# B&R Automation Studio project IecStringPrj (part 2)

#### test_float.c - Test IecStringFloat
```c
#include <UnitTest.h>
#include <IecString.h>
#include <string.h>
#include <stdint.h>
#include <float.h>

#define SAMPLE_SIZE 81
#define FULL_PRECISION 6
#define DEFAULT_WIDTH 0

_TEST test_float_variable(void) {
    char a[SAMPLE_SIZE];
    float value;
    int32_t status;

    value = 12e34f;

    status = IecStringFloat(a, sizeof(a), value,
                            DEFAULT_WIDTH, FULL_PRECISION, IECSTRING_FLAG_NONE);

    TEST_ASSERT_EQUAL_STRING("1.200000e+35", a);
    TEST_ASSERT_EQUAL_INT(IECSTRING_ERROR_NONE, status);

    TEST_DONE;
}

_TEST test_float_literal(void) {
    char a[SAMPLE_SIZE];
    int32_t status;

    status = IecStringFloat(a, sizeof(a), 12e34f,
                            DEFAULT_WIDTH, FULL_PRECISION, IECSTRING_FLAG_NONE);

    TEST_ASSERT_EQUAL_STRING("1.200000e+35", a);
    TEST_ASSERT_EQUAL_INT(IECSTRING_ERROR_NONE, status);

    TEST_DONE;
}

_TEST test_float_exponent_p5(void) {
    char a[SAMPLE_SIZE];
    int32_t status;

    status = IecStringFloat(a, sizeof(a), 123456.7f,
                            DEFAULT_WIDTH, FULL_PRECISION, IECSTRING_FLAG_NONE);

    TEST_ASSERT_EQUAL_STRING("123456.700000", a);
    TEST_ASSERT_EQUAL_INT(IECSTRING_ERROR_NONE, status);

    TEST_DONE;
}

_TEST test_float_exponent_p4(void) {
    char a[SAMPLE_SIZE];
    int32_t status;

    status = IecStringFloat(a, sizeof(a), 12345.67f,
                            DEFAULT_WIDTH, FULL_PRECISION, IECSTRING_FLAG_NONE);

    TEST_ASSERT_EQUAL_STRING("12345.670000", a);
    TEST_ASSERT_EQUAL_INT(IECSTRING_ERROR_NONE, status);

    TEST_DONE;
}

_TEST test_float_exponent_p3(void) {
    char a[SAMPLE_SIZE];
    int32_t status;

    status = IecStringFloat(a, sizeof(a), 1234.567f,
                            DEFAULT_WIDTH, FULL_PRECISION, IECSTRING_FLAG_NONE);

    TEST_ASSERT_EQUAL_STRING("1234.567000", a);
    TEST_ASSERT_EQUAL_INT(IECSTRING_ERROR_NONE, status);

    TEST_DONE;
}

_TEST test_float_exponent_p2(void) {
    char a[SAMPLE_SIZE];
    int32_t status;

    status = IecStringFloat(a, sizeof(a), 123.4567f,
                            DEFAULT_WIDTH, FULL_PRECISION, IECSTRING_FLAG_NONE);

    TEST_ASSERT_EQUAL_STRING("123.456700", a);
    TEST_ASSERT_EQUAL_INT(IECSTRING_ERROR_NONE, status);

    TEST_DONE;
}

_TEST test_float_exponent_p1(void) {
    char a[SAMPLE_SIZE];
    int32_t status;

    status = IecStringFloat(a, sizeof(a), 12.34567f,
                            DEFAULT_WIDTH, FULL_PRECISION, IECSTRING_FLAG_NONE);

    TEST_ASSERT_EQUAL_STRING("12.345670", a);
    TEST_ASSERT_EQUAL_INT(IECSTRING_ERROR_NONE, status);

    TEST_DONE;
}

_TEST test_float_exponent_0(void) {
    char a[SAMPLE_SIZE];
    int32_t status;

    status = IecStringFloat(a, sizeof(a), 1.234567f,
                            DEFAULT_WIDTH, FULL_PRECISION, IECSTRING_FLAG_NONE);

    TEST_ASSERT_EQUAL_STRING("1.234567", a);
    TEST_ASSERT_EQUAL_INT(IECSTRING_ERROR_NONE, status);

    TEST_DONE;
}

_TEST test_float_exponent_n1(void) {
    char a[SAMPLE_SIZE];
    int32_t status;

    status = IecStringFloat(a, sizeof(a), 0.1234567f,
                            DEFAULT_WIDTH, FULL_PRECISION, IECSTRING_FLAG_NONE);

    /* Rounding */
    TEST_ASSERT_EQUAL_STRING("0.123457", a);
    TEST_ASSERT_EQUAL_INT(IECSTRING_ERROR_NONE, status);

    TEST_DONE;
}

_TEST test_float_exponent_n2(void) {
    char a[SAMPLE_SIZE];
    int32_t status;

    status = IecStringFloat(a, sizeof(a), 0.01234567f,
                            DEFAULT_WIDTH, FULL_PRECISION, IECSTRING_FLAG_NONE);

    /* Rounding */
    TEST_ASSERT_EQUAL_STRING("0.012346", a);
    TEST_ASSERT_EQUAL_INT(IECSTRING_ERROR_NONE, status);

    TEST_DONE;
}

_TEST test_float_exponent_n3(void) {
    char a[SAMPLE_SIZE];
    int32_t status;

    status = IecStringFloat(a, sizeof(a), 0.001234567f,
                            DEFAULT_WIDTH, FULL_PRECISION, IECSTRING_FLAG_NONE);

    /* Rounding */
    TEST_ASSERT_EQUAL_STRING("0.001235", a);
    TEST_ASSERT_EQUAL_INT(IECSTRING_ERROR_NONE, status);

    TEST_DONE;
}

_TEST test_float_exponent_n4(void) {
    char a[SAMPLE_SIZE];
    int32_t status;

    status = IecStringFloat(a, sizeof(a), 0.0001234567f,
                            DEFAULT_WIDTH, FULL_PRECISION, IECSTRING_FLAG_NONE);

    TEST_ASSERT_EQUAL_STRING("0.000123", a);
    TEST_ASSERT_EQUAL_INT(IECSTRING_ERROR_NONE, status);

    TEST_DONE;
}

_TEST test_float_exponent_n5(void) {
    char a[SAMPLE_SIZE];
    int32_t status;

    status = IecStringFloat(a, sizeof(a), 0.00001234567f,
                            DEFAULT_WIDTH, FULL_PRECISION, IECSTRING_FLAG_NONE);

    TEST_ASSERT_EQUAL_STRING("0.000012", a);
    TEST_ASSERT_EQUAL_INT(IECSTRING_ERROR_NONE, status);

    TEST_DONE;
}

_TEST test_float_exponent_n6(void) {
    char a[SAMPLE_SIZE];
    int32_t status;

    status = IecStringFloat(a, sizeof(a), 0.000001234567f,
                            DEFAULT_WIDTH, FULL_PRECISION, IECSTRING_FLAG_NONE);

    TEST_ASSERT_EQUAL_STRING("0.000001", a);
    TEST_ASSERT_EQUAL_INT(IECSTRING_ERROR_NONE, status);

    TEST_DONE;
}

_TEST test_float_rollover_p5(void) {
    char a[SAMPLE_SIZE];
    int32_t status;

    /* Float stored as 999999.9375 or 1000000.0 */
    status = IecStringFloat(a, sizeof(a), 999999.97f,
                            DEFAULT_WIDTH, FULL_PRECISION, IECSTRING_FLAG_NONE);

    TEST_ASSERT_EQUAL_STRING("1.000000e+06", a);
    TEST_ASSERT_EQUAL_INT(IECSTRING_ERROR_NONE, status);

    TEST_DONE;
}

_TEST test_float_rollover_p2(void) {
    char a[SAMPLE_SIZE];
    int32_t status;

    /* Float stored as 999.99993896484375 or 1000.0 */
    status = IecStringFloat(a, sizeof(a), 999.99997f,
                            DEFAULT_WIDTH, FULL_PRECISION, IECSTRING_FLAG_NONE);

    TEST_ASSERT_EQUAL_STRING("1000.000000", a);
    TEST_ASSERT_EQUAL_INT(IECSTRING_ERROR_NONE, status);

    TEST_DONE;
}

_TEST test_float_rollover_0(void) {
    char a[SAMPLE_SIZE];
    int32_t status;

    status = IecStringFloat(a, sizeof(a), 0.9999995f,
                            DEFAULT_WIDTH, FULL_PRECISION, IECSTRING_FLAG_NONE);

    TEST_ASSERT_EQUAL_STRING("1.000000", a);
    TEST_ASSERT_EQUAL_INT(IECSTRING_ERROR_NONE, status);

    TEST_DONE;
}

_TEST test_float_rollover_n3(void) {
    char a[SAMPLE_SIZE];
    int32_t status;

    status = IecStringFloat(a, sizeof(a), 0.0009995f,
                            DEFAULT_WIDTH, FULL_PRECISION, IECSTRING_FLAG_NONE);

    TEST_ASSERT_EQUAL_STRING("0.001000", a);
    TEST_ASSERT_EQUAL_INT(IECSTRING_ERROR_NONE, status);

    TEST_DONE;
}

_TEST test_float_rollover_n6(void) {
    char a[SAMPLE_SIZE];
    int32_t status;

    /* Float stored as 9.99999883788e-07 or 9.99999997475e-07 */
    status = IecStringFloat(a, sizeof(a), 9.9999995e-7f,
                            DEFAULT_WIDTH, FULL_PRECISION, IECSTRING_FLAG_NONE);

    TEST_ASSERT_EQUAL_STRING("1.000000e-06", a);
    TEST_ASSERT_EQUAL_INT(IECSTRING_ERROR_NONE, status);

    TEST_DONE;
}

_TEST test_float_p37_A(void) {
    char a[SAMPLE_SIZE];
    int32_t status;

    /* Float representation is 9.99999460968e+37 */
    status = IecStringFloat(a, sizeof(a), 9.999995e37f,
                            DEFAULT_WIDTH, FULL_PRECISION, IECSTRING_FLAG_NONE);

    TEST_ASSERT_EQUAL_STRING("9.999995e+37", a);
    TEST_ASSERT_EQUAL_INT(IECSTRING_ERROR_NONE, status);

    TEST_DONE;
}

_TEST test_float_p37_B(void) {
    char a[SAMPLE_SIZE];
    int32_t status;

    /* Float representation is 9.99999866617e+37 or 9.99999968029e+37 */
    status = IecStringFloat(a, sizeof(a), 9.999999e37f,
                            DEFAULT_WIDTH, FULL_PRECISION, IECSTRING_FLAG_NONE);

    TEST_ASSERT_EQUAL_STRING("9.999999e+37", a);
    TEST_ASSERT_EQUAL_INT(IECSTRING_ERROR_NONE, status);

    TEST_DONE;
}

_TEST test_float_precision_3(void) {
    char a[SAMPLE_SIZE];
    int32_t status;

    status = IecStringFloat(a, sizeof(a), 0.123456f,
                            DEFAULT_WIDTH, 3, IECSTRING_FLAG_NONE);

    TEST_ASSERT_EQUAL_STRING("0.123", a);
    TEST_ASSERT_EQUAL_INT(IECSTRING_ERROR_NONE, status);

    TEST_DONE;
}

_TEST test_float_precision_3_round(void) {
    char a[SAMPLE_SIZE];
    int32_t status;

    status = IecStringFloat(a, sizeof(a), 0.99951f,
                            DEFAULT_WIDTH, 3, IECSTRING_FLAG_NONE);

    TEST_ASSERT_EQUAL_STRING("1.000", a);
    TEST_ASSERT_EQUAL_INT(IECSTRING_ERROR_NONE, status);

    TEST_DONE;
}

_TEST test_float_precision_0(void) {
    char a[SAMPLE_SIZE];
    int32_t status;

    status = IecStringFloat(a, sizeof(a), 123.456f,
                            DEFAULT_WIDTH, 0, IECSTRING_FLAG_NONE);

    TEST_ASSERT_EQUAL_STRING("123", a);
    TEST_ASSERT_EQUAL_INT(IECSTRING_ERROR_NONE, status);

    TEST_DONE;
}

_TEST test_float_precision_0_round(void) {
    char a[SAMPLE_SIZE];
    int32_t status;

    status = IecStringFloat(a, sizeof(a), 1.5f,
                            DEFAULT_WIDTH, 0, IECSTRING_FLAG_NONE);

    TEST_ASSERT_EQUAL_STRING("2", a);
    TEST_ASSERT_EQUAL_INT(IECSTRING_ERROR_NONE, status);

    TEST_DONE;
}

_TEST test_float_precision_0_notation(void) {
    char a[SAMPLE_SIZE];
    int32_t status;

    status = IecStringFloat(a, sizeof(a), 1.5e20f,
                            DEFAULT_WIDTH, 0, IECSTRING_FLAG_NONE);

    TEST_ASSERT_EQUAL_STRING("2e+20", a);
    TEST_ASSERT_EQUAL_INT(IECSTRING_ERROR_NONE, status);

    TEST_DONE;
}

_TEST test_float_max(void) {
    char a[SAMPLE_SIZE];
    int32_t status;

    status = IecStringFloat(a, sizeof(a), FLT_MAX,
                            DEFAULT_WIDTH, FULL_PRECISION, IECSTRING_FLAG_NONE);

    TEST_ASSERT_EQUAL_STRING("3.402823e+38", a);
    TEST_ASSERT_EQUAL_INT(IECSTRING_ERROR_NONE, status);

    TEST_DONE;
}

_TEST test_float_min(void) {
    char a[SAMPLE_SIZE];
    int32_t status;

    status = IecStringFloat(a, sizeof(a), FLT_MIN,
                            DEFAULT_WIDTH, FULL_PRECISION, IECSTRING_FLAG_NONE);

    TEST_ASSERT_EQUAL_STRING("1.175494e-38", a);
    TEST_ASSERT_EQUAL_INT(IECSTRING_ERROR_NONE, status);

    TEST_DONE;
}

_TEST test_float_zero(void) {
    char a[SAMPLE_SIZE];
    int32_t status, raw_value = 0;
    float value;

    memcpy(&value, &raw_value, 4);

    status = IecStringFloat(a, sizeof(a), value,
                            DEFAULT_WIDTH, FULL_PRECISION, IECSTRING_FLAG_NONE);

    TEST_ASSERT_EQUAL_STRING("0", a);
    TEST_ASSERT_EQUAL_INT(IECSTRING_ERROR_NONE, status);

    TEST_DONE;
}

_TEST test_float_negative_zero(void) {
    char a[SAMPLE_SIZE];
    int32_t status, raw_value = 0;
    float value;

    raw_value |= 1 << 31;
    memcpy(&value, &raw_value, 4);

    status = IecStringFloat(a, sizeof(a), value,
                            DEFAULT_WIDTH, FULL_PRECISION, IECSTRING_FLAG_NONE);

    TEST_ASSERT_EQUAL_STRING("-0", a);
    TEST_ASSERT_EQUAL_INT(IECSTRING_ERROR_NONE, status);

    TEST_DONE;
}

_TEST test_float_infinity(void) {
    char a[SAMPLE_SIZE];
    int32_t status, raw_value = 0;
    float value;

    raw_value |= 0xff << 23;
    memcpy(&value, &raw_value, 4);

    status = IecStringFloat(a, sizeof(a), value,
                            DEFAULT_WIDTH, FULL_PRECISION, IECSTRING_FLAG_NONE);

    TEST_ASSERT_EQUAL_STRING("inf", a);
    TEST_ASSERT_EQUAL_INT(IECSTRING_ERROR_NONE, status);

    TEST_DONE;
}

_TEST test_float_negative_infinity(void) {
    char a[SAMPLE_SIZE];
    int32_t status, raw_value = 0;
    float value;

    raw_value |= (1 << 31) + (0xff << 23);
    memcpy(&value, &raw_value, 4);

    status = IecStringFloat(a, sizeof(a), value,
                            DEFAULT_WIDTH, FULL_PRECISION, IECSTRING_FLAG_NONE);

    TEST_ASSERT_EQUAL_STRING("-inf", a);
    TEST_ASSERT_EQUAL_INT(IECSTRING_ERROR_NONE, status);

    TEST_DONE;
}

_TEST test_float_not_a_number(void) {
    char a[SAMPLE_SIZE];
    int32_t status, raw_value = 0;
    float value;

    raw_value |= (0xff << 23) + 1;
    memcpy(&value, &raw_value, 4);

    status = IecStringFloat(a, sizeof(a), value,
                            DEFAULT_WIDTH, FULL_PRECISION, IECSTRING_FLAG_NONE);

    TEST_ASSERT_EQUAL_STRING("NaN", a);
    TEST_ASSERT_EQUAL_INT(IECSTRING_ERROR_NONE, status);

    TEST_DONE;
}

_TEST test_float_size_zero(void) {
    char a[SAMPLE_SIZE];
    int32_t status;

    strcpy(a, "abc");
    status = IecStringFloat(a, 0, 123.0f,
                            DEFAULT_WIDTH, FULL_PRECISION, IECSTRING_FLAG_NONE);

    TEST_ASSERT_EQUAL_STRING("abc", a);
    TEST_ASSERT_EQUAL_INT(IECSTRING_ERROR_SIZE_ZERO, status);

    TEST_DONE;
}

_TEST test_float_size_one(void) {
    char a[SAMPLE_SIZE];
    int32_t status;

    strcpy(a, "abc");
    status = IecStringFloat(a, 1, 123.0f,
                            DEFAULT_WIDTH, FULL_PRECISION, IECSTRING_FLAG_NONE);

    TEST_ASSERT_EQUAL_STRING("", a);
    TEST_ASSERT_EQUAL_INT(IECSTRING_ERROR_SIZE_INVALID, status);

    TEST_DONE;
}

_TEST test_float_size_invalid(void) {
    char a[SAMPLE_SIZE];
    int32_t status;

    strcpy(a, "abc");
    /* Requires size of 11 for full precision 123.000000 */
    status = IecStringFloat(a, 6, 123.0f,
                            DEFAULT_WIDTH, FULL_PRECISION, IECSTRING_FLAG_NONE);

    TEST_ASSERT_EQUAL_STRING("", a);
    TEST_ASSERT_EQUAL_INT(IECSTRING_ERROR_SIZE_INVALID, status);

    TEST_DONE;
}

_TEST test_float_null(void) {
    int32_t status;

    status = IecStringFloat(NULL, SAMPLE_SIZE, 123.0f,
                            DEFAULT_WIDTH, FULL_PRECISION, IECSTRING_FLAG_NONE);

    TEST_ASSERT_EQUAL_INT(IECSTRING_ERROR_NULL, status);

    TEST_DONE;
}

UNITTEST_FIXTURES(fixtures) {
    new_TestFixture("IecStringFloat from variable", test_float_variable),
    new_TestFixture("IecStringFloat from literal", test_float_literal),
    new_TestFixture("IecStringFloat exponent +5", test_float_exponent_p5),
    new_TestFixture("IecStringFloat exponent +4", test_float_exponent_p4),
    new_TestFixture("IecStringFloat exponent +3", test_float_exponent_p3),
    new_TestFixture("IecStringFloat exponent +2", test_float_exponent_p2),
    new_TestFixture("IecStringFloat exponent +1", test_float_exponent_p1),
    new_TestFixture("IecStringFloat exponent  0", test_float_exponent_0),
    new_TestFixture("IecStringFloat exponent -1", test_float_exponent_n1),
    new_TestFixture("IecStringFloat exponent -2", test_float_exponent_n2),
    new_TestFixture("IecStringFloat exponent -3", test_float_exponent_n3),
    new_TestFixture("IecStringFloat exponent -4", test_float_exponent_n4),
    new_TestFixture("IecStringFloat exponent -5", test_float_exponent_n5),
    new_TestFixture("IecStringFloat exponent -6", test_float_exponent_n6),
    new_TestFixture("IecStringFloat rollover +5", test_float_rollover_p5),
    new_TestFixture("IecStringFloat rollover +2", test_float_rollover_p2),
    new_TestFixture("IecStringFloat rollover  0", test_float_rollover_0),
    new_TestFixture("IecStringFloat rollover -3", test_float_rollover_n3),
    new_TestFixture("IecStringFloat rollover -6", test_float_rollover_n6),
    new_TestFixture("IecStringFloat precision 3", test_float_precision_3),
    new_TestFixture("IecStringFloat precision 3 round",
                    test_float_precision_3_round),
    new_TestFixture("IecStringFloat exponent +37 test A", test_float_p37_A),
    new_TestFixture("IecStringFloat exponent +37 test B", test_float_p37_B),
    new_TestFixture("IecStringFloat precision 0", test_float_precision_0),
    new_TestFixture("IecStringFloat precision 0 round",
                    test_float_precision_0_round),
    new_TestFixture("IecStringFloat precision 0 scientific notation",
                    test_float_precision_0_notation),
    new_TestFixture("IecStringFloat max", test_float_max),
    new_TestFixture("IecStringFloat min", test_float_min),
    new_TestFixture("IecStringFloat zero", test_float_zero),
    new_TestFixture("IecStringFloat negative zero", test_float_negative_zero),
    new_TestFixture("IecStringFloat infinity", test_float_infinity),
    new_TestFixture("IecStringFloat negative infinity",
                    test_float_negative_infinity),
    new_TestFixture("IecStringFloat not a number", test_float_not_a_number),
    new_TestFixture("IecStringFloat size zero", test_float_size_zero),
    new_TestFixture("IecStringFloat size one", test_float_size_one),
    new_TestFixture("IecStringFloat size invalid", test_float_size_invalid),
    new_TestFixture("IecStringFloat null", test_float_null)
};

UNITTEST_CALLER_TEST(float_set, "IecStringFloat test set", fixtures);
```

#### test_date_time.c - Test IecStringDateTime
```c
#include <UnitTest.h>
#include <IecString.h>
#include <astime.h>
#include <string.h>
#include <stdint.h>

#define SAMPLE_SIZE 81

DTStructure value = {
    .year = 2024,
    .month = 1,
    .day = 9,
    .wday = 2,
    .hour = 13,
    .minute = 4,
    .second = 9,
    .millisec = 55
};

_TEST test_date_time_default(void) {
    char a[SAMPLE_SIZE];
    int32_t status;

    status = IecStringDateTime(a, sizeof(a), &value, NULL);

    TEST_ASSERT_EQUAL_STRING("2024-01-09 13:04", a);
    TEST_ASSERT_EQUAL_INT(IECSTRING_ERROR_NONE, status);

    TEST_DONE;
}

_TEST test_date_time_formal_date(void) {
    char a[SAMPLE_SIZE];
    int32_t status;

    status = IecStringDateTime(a, sizeof(a), &value, "dddd, MMMM d, yyyy");

    TEST_ASSERT_EQUAL_STRING("Tuesday, January 9, 2024", a);
    TEST_ASSERT_EQUAL_INT(IECSTRING_ERROR_NONE, status);

    TEST_DONE;
}

UNITTEST_FIXTURES(fixtures) {
    new_TestFixture("IecStringDateTime default", test_date_time_default),
    new_TestFixture("IecStringDateTime formal date", test_date_time_formal_date)
};

UNITTEST_CALLER_TEST(date_time_set, "IecStringDateTime test set", fixtures);
```

#### test_integer.c - not listed in the package file held
```c
#include <UnitTest.h>
#include <IecString.h>
#include <string.h>
#include <stdint.h>

_TEST test_integer_zeros(void) {
    char a[81];
    int32_t number, status;

    number = 1234;

    status = IecStringInteger(a, sizeof(a), number, 6, '0');

    TEST_ASSERT_EQUAL_STRING("001234", a);
    TEST_ASSERT_EQUAL_INT(0, status);

    TEST_DONE;
}

_TEST test_integer_spaces(void) {
    char a[81];
    int32_t number, status;

    number = -5678;

    status = IecStringInteger(a, sizeof(a), number, 6, ' ');

    /* Width includes sign */
    TEST_ASSERT_EQUAL_STRING("- 5678", a);
    TEST_ASSERT_EQUAL_INT(0, status);

    /* Defaults to spaces */
    status = IecStringInteger(a, sizeof(a), number, 6, 0);

    TEST_ASSERT_EQUAL_STRING("- 5678", a);
    TEST_ASSERT_EQUAL_INT(0, status);

    TEST_DONE;
}

_TEST test_integer_tilde(void) {
    char a[81];
    int32_t number, status;

    number = 9012;

    status = IecStringInteger(a, sizeof(a), number, 6, '~');

    TEST_ASSERT_EQUAL_STRING("~~9012", a);
    TEST_ASSERT_EQUAL_INT(0, status);

    TEST_DONE;
}

_TEST test_integer_max(void) {
    char a[81];
    int32_t number, status;

    number = INT32_MAX;

    status = IecStringInteger(a, sizeof(a), number, 0, '0');

    TEST_ASSERT_EQUAL_STRING("2147483647", a);
    TEST_ASSERT_EQUAL_INT(0, status);

    TEST_DONE;
}

_TEST test_integer_min(void) {
    char a[81];
    int32_t number, status;

    number = INT32_MIN;

    status = IecStringInteger(a, sizeof(a), number, 0, '0');

    TEST_ASSERT_EQUAL_STRING("-2147483648", a);
    TEST_ASSERT_EQUAL_INT(0, status);

    TEST_DONE;
}

_TEST test_integer_size(void) {
    char a[6];
    int32_t number, status;

    strcpy(a, "abc");
    number = 123456;

    status = IecStringInteger(a, sizeof(a), number, 0, '0');

    TEST_ASSERT_EQUAL_STRING("abc", a);
    TEST_ASSERT_EQUAL_INT(IECSTRING_ERROR_SIZE, status);

    TEST_DONE;
}

_TEST test_integer_null(void) {
    int32_t number, status;

    number = 123456;

    status = IecStringInteger(NULL, 7, number, 0, '0');

    TEST_ASSERT_EQUAL_INT(IECSTRING_ERROR_NULL, status);

    TEST_DONE;
}

UNITTEST_FIXTURES(fixtures) {
    new_TestFixture("IecStringInteger zeros", test_integer_zeros),
    new_TestFixture("IecStringInteger spaces", test_integer_spaces),
    new_TestFixture("IecStringInteger tilde", test_integer_tilde),
    new_TestFixture("IecStringInteger max", test_integer_max),
    new_TestFixture("IecStringInteger min", test_integer_min),
    new_TestFixture("IecStringInteger size error", test_integer_size),
    new_TestFixture("IecStringInteger null error", test_integer_null)
};

UNITTEST_CALLER_TEST (padint_set, "IecStringInteger test set", fixtures);
```

### Program Logical/Source/UnitTest/TestFloat (ANSIC)

#### Variables.var
```iecst
VAR
	FloatValue : REAL;
	PromotionToDouble : LREAL;
	LibFloatText : STRING[80];
	BrsFloatText : STRING[80];
	FloatRaw : UDINT;
	TestInfinity : BOOL;
	TestNotANumber : BOOL;
	Log10Value : REAL;
	Precision : USINT;
END_VAR
```

#### Main.c
```c
#include <bur/plc.h>
#include <Variablesvar.h>
#include <IecString.h>
#include <AsBrStr.h>
#include <stdint.h>
#include <math.h>

void _CYCLIC ProgramCyclic(void) {
    IecStringFloat(LibFloatText, sizeof(LibFloatText), FloatValue);
    brsftoa(FloatValue, (uint32_t)BrsFloatText);
    PromotionToDouble = FloatValue;
    FloatRaw = *(uint32_t*)&FloatValue;

    if (TestInfinity) {
        TestInfinity = 0;
        FloatValue *= 1.0e38f;
    }

    if (TestNotANumber) {
        TestNotANumber = 0;
        FloatValue /= 0.0f;
    }

    Log10Value = log10f(FloatValue);
}
```

### Program Logical/Source/UnitTest/TestCopy (ANSIC)

#### Variables.var
```iecst
VAR
	String1 : STRING[80];
	String2 : STRING[80];
	MySize : UDINT := 6;
	MyStatus : DINT;
END_VAR
```

#### Main.c
```c
#include <bur/plc.h>
#include <Variablesvar.h>
#include <IecString.h>

void _CYCLIC ProgramCyclic(void) {
    MyStatus = IecStringCopy(String1, MySize, String2);
}
```

### Program Logical/Source/UnitTest/TestDT (IEC)

#### Variables.var
```iecst
VAR
	DateAndTimeData : DTStructure;
	String1 : STRING[80];
	String2 : STRING[80];
	GetDateAndTime : DTStructureGetTime;
END_VAR
```

#### Main.st
```iecst
PROGRAM _INIT
	GetDateAndTime(enable := TRUE, pDTStructure := ADR(DateAndTimeData));
END_PROGRAM

PROGRAM _CYCLIC
	IecStringDateTime(String1, SIZEOF(String1), DateAndTimeData, String2);
END_PROGRAM
```

### Program Logical/Source/Example/ExSplit (IEC)

#### Variables.var
```iecst
(*Command*)
VAR
	Run : BOOL;
END_VAR
(*Data*)
VAR
	Source : STRING[80];
	SourceReference : REFERENCE TO STRING[80];
	NextAddress : UDINT;
	Delimeters : STRING[80];
	Words : ARRAY[0..9] OF STRING[80];
	Index : USINT;
END_VAR
```

#### Main.st
```iecst
PROGRAM _INIT

	Source := 'The quick brown fox jumps over the lazy dog';
	Delimeters := ' ';

END_PROGRAM

PROGRAM _CYCLIC

	IF Run THEN
		Run := FALSE;

		brsmemset(ADR(Words), 0, SIZEOF(Words));
		Index := 0;

		SourceReference ACCESS ADR(Source);
		REPEAT
			IecStringSplit(Words[Index], SIZEOF(Words[Index]), SourceReference, Delimeters, NextAddress);
			SourceReference ACCESS NextAddress;
			Index := Index + 1;
		UNTIL
			Index >= SIZEOF(Words) / SIZEOF(Words[0]) OR NextAddress = 0
		END_REPEAT
		SourceReference ACCESS ADR(Source);
	END_IF

END_PROGRAM
```

### Program Logical/Source/Performance/ACopy1C (ANSIC) - Performance of strcpy

#### Main.c
```c
#include <bur/plc.h>
#include <string.h>

void _CYCLIC ProgramCyclic(void)
{
    char a[81];
    int i;
    for (i = 0; i < 100; i++)
        strcpy(a, "This is a test of string copy performance across multiple libraries.");
}
```

### Program Logical/Source/Performance/ACopy2Iec (IEC) - Performacce of IEC string assignment

#### Variables.var
```iecst
VAR
	i : INT;
	a : STRING[254];
	b : STRING[254] := '0123456789abcdefghij0123456789abcdefghij0123456789abcdefghij0123456789abcdefghij';
END_VAR
```

#### Main.st
```iecst
(* 100 calls to copy 80 characters *)
PROGRAM _CYCLIC
	FOR i := 0 TO 99 DO
		a := b;
	END_FOR
END_PROGRAM
```

### Program Logical/Source/Performance/ACopy3Brs (ANSIC) - Performance of brsstrcpy

#### Main.c
```c
#include <bur/plc.h>
#include <AsBrStr.h>

char a[255];
int i;

/* 100 calls to copy 80 characters */
void _CYCLIC ProgramCyclic(void)
{
    for (i = 0; i < 100; i++)
    {
        brsstrcpy((unsigned long)a,
                  (unsigned long)"0123456789abcdefghij0123456789abcdefghij"
                                 "0123456789abcdefghij0123456789abcdefghij");
    }
}
```

### Program Logical/Source/Performance/ACopy4Lib (ANSIC) - Performance of IecStringCopy

#### Main.c
```c
#include <bur/plc.h>
#include <IecString.h>

char a[255];
int i;

/* 100 calls to copy 80 characters */
void _CYCLIC ProgramCyclic(void)
{
    for (i = 0; i < 100; i++)
    {
        IecStringCopy(a, sizeof(a), "0123456789abcdefghij0123456789abcdefghij"
                                    "0123456789abcdefghij0123456789abcdefghij");
    }
}
```

### Program Logical/Source/Performance/BCat1C (ANSIC) - Performance of strcat

#### Main.c
```c
#include <bur/plc.h>
#include <string.h>

char a[255] = "Hello World! 1234567890.";
int i;

void _CYCLIC ProgramCyclic(void) {
    for (i = 0; i < 100; i++) {
        a[24] = '\0';
        strcat(a, " The quick brown fox jumps over the lazy dog.");
    }
}
```

### Program Logical/Source/Performance/BCat2Iec (IEC) - Performance of CONCAT

#### Variables.var
```iecst
VAR
	i : INT;
	a : STRING[255];
END_VAR
```

#### Main.st
```iecst
(* 100 calls to concatenate 80 characters to length of 80 *)
PROGRAM _CYCLIC
	FOR i := 0 TO 99 DO
		a := CONCAT('0123456789abcdefghij0123456789abcdefghij0123456789abcdefghij0123456789abcdefghij', '0123456789abcdefghij0123456789abcdefghij0123456789abcdefghij0123456789abcdefghij');
	END_FOR
END_PROGRAM
```

### Program Logical/Source/Performance/BCat3Brs (ANSIC) - Performance of brsstrcat

#### Main.c
```c
#include <bur/plc.h>
#include <AsBrStr.h>
#include <stdint.h>

char a[81] = "Hello World! 1234567890.";
int i;

void _CYCLIC ProgramCyclic(void) {
    for (i = 0; i < 100; i++) {
        a[24] = '\0';
        brsstrcat((uint32_t)a, (uint32_t)" The quick brown fox jumps over the lazy dog.");
    }
}
```

### Program Logical/Source/Performance/BCat4Lib (ANSIC) - Performance of IecStringConcat

#### Main.c
```c
#include <bur/plc.h>
#include <IecString.h>

char a[255] = "0123456789abcdefghij0123456789abcdefghij"
              "0123456789abcdefghij0123456789abcdefghij";
int i;

/* 100 calls to concatenate 80 characters to length of 80 */
void _CYCLIC ProgramCyclic(void)
{
    for (i = 0; i < 100; i++)
    {
        a[80] = '\0';
        IecStringConcat(a, sizeof(a),
                        "0123456789abcdefghij0123456789abcdefghij"
                        "0123456789abcdefghij0123456789abcdefghij");
    }
}
```

### Program Logical/Source/Performance/EDec2Iec (IEC) - Performance of DINT_TO_STRING

#### Variables.var
```iecst
VAR
	i : INT;
	number : DINT := -2001001001;
	a : STRING[20];
END_VAR
```

#### Main.st
```iecst
(* 100 calls to convert integer to string *)
PROGRAM _CYCLIC
	FOR i := 0 TO 99 DO
		a := DINT_TO_STRING(number);
	END_FOR
END_PROGRAM
```

### Program Logical/Source/Performance/EDec3Brs (ANSIC) - Performance of brsitoa

#### Main.c
```c
#include <bur/plc.h>
#include <AsBrStr.h>

char a[21];
int i;
const signed long number = -2001001001;

void _CYCLIC ProgramCyclic(void) {
    for (i = 0; i < 100; i++)
        brsitoa(number, (unsigned long)a);
}
```

### Program Logical/Source/Performance/EDec4Lib (ANSIC) - Performance of IecStringDecimal

#### Main.c
```c
#include <bur/plc.h>
#include <IecString.h>

char a[21];
int i;
const signed long number = -2001001001;

void _CYCLIC ProgramCyclic(void) {
    for (i = 0; i < 100; i++)
        IecStringDecimal(a, sizeof(a), number, 5, '0', 0);
}
```

### Program Logical/Source/Performance/FFp2Iec (IEC) - Performance of AsIecCon's REAL_TO_STRING

#### Main.st
```iecst
(* 100 calls to convert float to string *)
PROGRAM _CYCLIC
	FOR i := 0 TO 99 DO
		a := REAL_TO_STRING(123.456e-23);
	END_FOR
END_PROGRAM
```

### Program Logical/Source/Performance/FFp3Brs (ANSIC) - Performance of AsBrStr's brsftoa

#### Main.c
```c
#include <bur/plc.h>
#include <AsBrStr.h>

char a[81];
int i;

/* 100 calls to convert float to string */
void _CYCLIC ProgramCyclic(void)
{
    for (i = 0; i < 100; i++)
        brsftoa(123.456e-23f, (unsigned long)a);
}
```

### Program Logical/Source/Performance/FFp4Lib (ANSIC) - Performance of IecStringFloat

#### Main.c
```c
#include <bur/plc.h>
#include <IecString.h>

char a[81];
int i;

/* 100 calls to convert float to string */
void _CYCLIC ProgramCyclic(void)
{
    for (i = 0; i < 100; i++)
        IecStringFloat(a, sizeof(a), 123.456e-23f, 0, 6, IECSTRING_FLAG_NONE);
}
```

### Program Logical/Source/Performance/ACopy2Br

#### Main.c
```c
#include <bur/plc.h>
#include <stdint.h>
#include <AsBrStr.h>

void _CYCLIC ProgramCyclic(void)
{
    char a[81];
    int i;
    for (i = 0; i < 100; i++)
        brsstrcpy((uint32_t)a, (uint32_t)"This is a test of string copy performance across multiple libraries");
}
```

### Program Logical/Source/Performance/ACopy3IS (ANSIC)

#### Main.c - Init, cyclic, exit code
```c
#include <bur/plc.h>
#include <IecString.h>

void _CYCLIC ProgramCyclic(void)
{
    char a[81];
    int i;
    for (i = 0; i < 100; i++)
        IecStringCopy(a, sizeof(a), "This is a test of string copy performance");
}
```

### Program Logical/Source/Performance/BCat2Br

#### Main.c
```c
#include <bur/plc.h>
#include <AsBrStr.h>
#include <stdint.h>

void _CYCLIC ProgramCyclic(void)
{
    char a[81] = "Hello World! 1234567890.";
    int i;
    for (i = 0; i < 100; i++) {
        a[19] = '\0';
        brsstrcat((uint32_t)a, (uint32_t)" The quick brown fox jumps over the lazy dog.");
    }
}
```

### Program Logical/Source/Performance/BCat3IS

#### Main.c
```c
#include <bur/plc.h>
#include <IecString.h>

void _CYCLIC ProgramCyclic(void)
{
    char a[81] = "Hello World! 1234567890.";
    int i;
    for (i = 0; i < 100; i++) {
        a[19] = '\0';
        IecStringConcat(a, sizeof(a), " The quick brown fox jumps over the lazy dog.");
    }
}
```

### Program Logical/Source/Performance/CPUCopy

#### Main.c
```c
#include <bur/plc.h>
#include <bur/plctypes.h>
#include <IecString.h>
#include <AsBrStr.h>
#include <string.h>

_LOCAL UINT count _VAR_INIT(100);

void _CYCLIC ProgramCyclic(void)
{
    char a[81], b[81];
    DINT i;
    IecStringCopy(b, sizeof(b), "This is a test of string copy performance");

    /* Test strcpy */
    for (i = 0; i < count; i++)
        strcpy(a, b);

    /* Test brsstrcpy */
    for (i = 0; i < count; i++)
        brsstrcpy((UDINT)a, (UDINT)b);

    /* Test IecStringCopy */
    for (i = 0; i < count; i++)
        IecStringCopy(a, sizeof(a), b);
}
```

### Program Logical/Source/Performance/CPUDecimal

#### Main.c
```c
#include <bur/plc.h>
#include <bur/plctypes.h>
#include <IecString.h>
#include <AsBrStr.h>

_LOCAL UINT count _VAR_INIT(100);

void _CYCLIC ProgramCyclic(void)
{
    char a[21];
    DINT i, number = -2001001001;

    /* Test brsitoa */
    for (i = 0; i < count; i++)
        brsitoa(number, (UDINT)a);

    /* Test IecStringInteger */
    for (i = 0; i < count; i++)
        IecStringInteger(a, sizeof(a), number, 5, '0');
}
```

### Program Logical/Source/Performance/EDec2Br

#### Main.c
```c
#include <bur/plc.h>
#include <stdint.h>
#include <AsBrStr.h>

void _CYCLIC ProgramCyclic(void)
{
    char a[21];
    int32_t i, number = -2001001001;
    for (i = 0; i < 100; i++)
        brsitoa(number, (UDINT)a);
}
```

### Program Logical/Source/Performance/PerfBase

#### Main.c
```c
#include <bur/plc.h>

void _CYCLIC ProgramCyclic(void)
{
    char a[81], b[81];
    int i;
    for (i = 0; i < 100; i++)
        i;
}
```

### Program Logical/Source/Performance/PerfBrCopy

#### Main.c
```c
#include <bur/plc.h>
#include <bur/plctypes.h>
#include <AsBrStr.h>

void _CYCLIC ProgramCyclic(void)
{
    char a[81];
    int i;
    for (i = 0; i < 100; i++)
        brsstrcpy((UDINT)a, "This is a test of string copy performance");
}
```

### Program Logical/Source/Performance/PerfISDec

#### Main.c
```c
#include <bur/plc.h>
#include <stdint.h>
#include <IecString.h>

void _CYCLIC ProgramCyclic(void)
{
    char a[21];
    int32_t i, number = -2001001001;
    for (i = 0; i < 100; i++)
        IecStringInteger(a, sizeof(a), number, 5, '0');
}
```

### Program Logical/Source/Compare/CFloat (ANSIC) - Test floating point values

#### Main.c
```c
#include <bur/plc.h>
#include <stdint.h>
#include <string.h>

_LOCAL float number;
_LOCAL uint32_t data, sign, exponent, fraction;
_LOCAL int32_t int_cast;

void _CYCLIC ProgramCyclic(void)
{
    memcpy(&data, &number, sizeof(data));
    sign = (data >> 31) & 0x1;
    exponent = (data >> 23) & 0xFF;
    fraction = data & 0x7FFFFF;
    int_cast = (int)number;
}
```

### Program Logical/Source/Compare/Float (IEC)

#### Variables.var
```iecst
VAR
	FloatValue : REAL;
	DoublePromotionValue : LREAL;
	LibFloatText : STRING[80];
	BrsFloatText : STRING[80];
END_VAR
```

#### Main.st
```iecst
PROGRAM _CYCLIC
	DoublePromotionValue := FloatValue;
	IecStringFloat(LibFloatText, SIZEOF(LibFloatText), FloatValue);
	brsftoa(FloatValue, ADR(BrsFloatText));
END_PROGRAM
```

### Program Logical/Source/Compare/BrDecimal

#### Variables.var
```iecst
VAR
	Number : DINT;
	NumberText : STRING[14];
	NumberData : REFERENCE TO ARRAY[0..14] OF USINT;
END_VAR
```

#### Main.st
```iecst
PROGRAM _CYCLIC

	brsitoa(Number, ADR(NumberText));
	NumberData ACCESS ADR(NumberText);

END_PROGRAM
```

### Program Logical/Source/Compare/BrFloat

#### Variables.var
```iecst
VAR
	Number : REAL;
	NumberText : STRING[14];
	NumberData : REFERENCE TO ARRAY[0..14] OF USINT;
END_VAR
```

#### Main.st
```iecst
PROGRAM _CYCLIC

	brsftoa(Number, ADR(NumberText));
	NumberData ACCESS ADR(NumberText);

END_PROGRAM
```

### Program Logical/Source/Sample/IECST (IEC)

#### Variables.var
```iecst
(*IecStringCopy*)
VAR
	Source : STRING[10] := 'Program';
	Destination : STRING[5];
END_VAR
(*IecStringFormat*)
VAR
	FromattedString : STRING[80];
	FormatValues : IecStringFormatType;
END_VAR
(*IecStringInteger*)
VAR
	MyInteger : INT;
	PaddedInteger : STRING[80];
END_VAR
(*IecStringDateTime*)
VAR
	DateTimeString : STRING[80];
	FormatDateTime : STRING[80];
	DateTime : DTStructure;
	GetDateTime : DTStructureGetTime;
	CurrentDateTime : DTStructure;
END_VAR
(*Raw characters*)
VAR
	Raw1 : ARRAY[0..10] OF USINT;
	Raw2 : ARRAY[0..10] OF USINT;
	ReferenceString1 : REFERENCE TO STRING[10];
	ReferenceString2 : REFERENCE TO STRING[10];
END_VAR
```

#### Main.st
```iecst
PROGRAM _INIT

	FormatValues.b[0] := TRUE;
	FormatValues.f[0] := 12.34;
	FormatValues.i[0] := 33;
	FormatValues.s[0] := 'All Clear';

END_PROGRAM

PROGRAM _CYCLIC

	IecStringCopy(Destination,
		SIZEOF(Destination),
		Source);

	ReferenceString1 ACCESS ADR(Raw1);
	ReferenceString2 ACCESS ADR(Raw2);
	IecStringCopy(ReferenceString1, SIZEOF(ReferenceString1), ReferenceString2);

	IecStringFormat(FromattedString,
		SIZEOF(FromattedString),
		'Error: %b, Temp: %f C, Step: %i, Message: %s',
		FormatValues);

	IecStringInteger(PaddedInteger,
		SIZEOF(PaddedInteger),
		MyInteger,
		6,
		FALSE);

	GetDateTime(enable := TRUE, pDTStructure := ADR(CurrentDateTime));
	IecStringDateTime(DateTimeString, SIZEOF(DateTimeString), FormatDateTime, DateTime);

END_PROGRAM
```

### Program Logical/Source/Sample/Float (IEC)

#### Variables.var
```iecst
VAR
	String1 : STRING[80];
	Value : REAL;
	Width : USINT;
	Precision : USINT;
END_VAR
```

#### Main.st
```iecst
PROGRAM _CYCLIC

	IecStringFloat(String1, SIZEOF(String1), Value, Width, Precision, IECSTRING_FLAG_NONE);

END_PROGRAM
```

### Program Logical/Source/Sample/ExFloat

#### Variables.var
```iecst
VAR
	Float : REAL;
	FloatText : STRING[80];
END_VAR
```

#### Main.st
```iecst
PROGRAM _CYCLIC

	IecStringFloat(FloatText, SIZEOF(FloatText), Float);

END_PROGRAM
```

- IecStringText.csv (not shown)

- IecStringGenerate.py (not shown)

### Program Logical/CUsage

#### Variables.var
```iecst
VAR
	format : STRING[80];
	formatArgs : FormatStringArgumentsType;
	message : STRING[80];
	length : UDINT;
END_VAR
(*Pad whole number*)
VAR
	myNumber : DINT;
	number : STRING[20];
	digits : USINT;
	spaces : BOOL;
END_VAR
```

#### Main.c
```c
#include <bur/plctypes.h>

#ifdef _DEFAULT_INCLUDES
	#include <AsDefault.h>
#endif

#include <stdbool.h>
#include <string.h>

void _INIT ProgramInit(void)
{
	// Runtime values
	formatArgs.b[0] = false; // BOOL
	formatArgs.r[0] = 78.768; // LREAL
	formatArgs.i[0] = -2144327918; // DINT, e.g. Status ID
	strcpy(formatArgs.s[0], "INIT"); // STRING

	strcpy(format, "Status %b, Temp %r F, Code %i, State %s");

	myNumber = -1234;
	digits = 6;
	spaces = false;
}

void _CYCLIC ProgramCyclic(void)
{
	length = IecFormatString(message, sizeof(message), format, &formatArgs);

	IecPadNumber(myNumber, number, digits, spaces);
}

void _EXIT ProgramExit(void)
{

}
```

### Program Logical/IECST

#### Variables.var
```iecst
(*IecStringCopy*)
VAR
	Source : STRING[10] := 'Program';
	Destination : STRING[5];
END_VAR
(*IecStringFormat*)
VAR
	FromattedString : STRING[80];
	FormatValues : IecStringFormatType;
END_VAR
(*IecStringInteger*)
VAR
	MyInteger : INT;
	PaddedInteger : STRING[80];
END_VAR
(*IecStringDateTime*)
VAR
	DateTimeString : STRING[80];
	FormatDateTime : STRING[80];
END_VAR
```

#### Main.st
```iecst
PROGRAM _INIT

	FormatValues.b[0] := TRUE;
	FormatValues.f[0] := 12.34;
	FormatValues.i[0] := 33;
	FormatValues.s[0] := 'All Clear';

END_PROGRAM

PROGRAM _CYCLIC

	IecStringCopy(Destination,
		SIZEOF(Destination),
		Source);

	IecStringFormat(FromattedString,
		SIZEOF(FromattedString),
		'Error: %b, Temp: %f C, Step: %i, Message: %s',
		FormatValues);

	IecStringInteger(PaddedInteger,
		SIZEOF(PaddedInteger),
		MyInteger,
		6,
		FALSE);

	GetDateTime(enable := TRUE, pDTStructure := ADR(CurrentDateTime));
	IecStringDateTime(DateTimeString, SIZEOF(DateTimeString), FormatDateTime, DateTime);

END_PROGRAM
```

### Program Logical/Program

#### Variables.var
```iecst
VAR
	AllocationReturnStatus : UDINT;
	CyclicReturnStatus : UDINT;
	FreeReturnStatus : UDINT;
END_VAR
VAR CONSTANT
	STR_LEN_ALARM_MSG : USINT := 125;
END_VAR
VAR
	sConstructMessage : STRING[STR_LEN_ALARM_MSG];
	sFormattedMessage : STRING[STR_LEN_ALARM_MSG];
	MessageArguments : FormatStringArgumentsType;
	CmdLog : BOOL;
	EventID : DINT;
	ErrorCode : UINT;
END_VAR
```

#### Main.st
```iecst
(*******************************************************************************
 * Copyright: B&R Industrial Automation
 * Author:    Tyler Matijevich
 * Created:   September 27, 2020/11:19
********************************************************************************
 * Description: Example program for formatting string in IEC code and logging
 user entries in the logger
********************************************************************************)

PROGRAM _INIT

	// Allocates the FIFO buffer for the logger
	AllocationReturnStatus := BRSE_ARL_Alloc(ID := 1, Name := 'AppLog', LogbookSize := 10000, MessageSize := STR_LEN_ALARM_MSG, BufferedEntries := 25);

END_PROGRAM

PROGRAM _CYCLIC

	IF CmdLog THEN
		CmdLog := FALSE;

		// Construct and log message
		IecFormatString(ADR(sFormattedMessage), STR_LEN_ALARM_MSG, ADR(sConstructMessage), ADR(MessageArguments));
		EventID := ArEventLogMakeEventID(Severity := arEVENTLOG_SEVERITY_ERROR, Facility := 0, ErrorCode := ErrorCode);
		BRSE_ARL_Log(1, EventID, 'MyLog', sFormattedMessage);
	END_IF

	// Flush pending entries to the logbook
	CyclicReturnStatus := BRSE_ARL_Cyclic(ID := 1);

END_PROGRAM

PROGRAM _EXIT

	// Deallocate the FIFO buffer
	FreeReturnStatus := BRSE_ARL_Free(ID := 1);

END_PROGRAM
```

### Program Logical/Sample

#### Variables.var
```iecst
VAR
	Format : STRING[80];
	FormatArgs : FormatStringArgumentsType;
	Message : STRING[80];
	Size : UDINT;
	Length : UDINT;
END_VAR
(*AsBrStr test variables*)
VAR
	VarDint : DINT;
	sDint : STRING[80];
	ReturnDint : UINT;
	VarReal : REAL;
	sReal : STRING[80];
	ReturnReal : UINT;
END_VAR
(*IecPadNumber*)
VAR
	MyNumber : DINT;
	Number : STRING[20];
	Padding : USINT;
	Spaces : BOOL;
	Name1 : STRING[10];
	NameSpace : STRING[10];
	Name2 : STRING[20];
	Concat1 : STRING[10];
	ConcatSpace : STRING[10];
	Concat2 : STRING[20];
	CmdConcat : BOOL;
END_VAR
(*Find and replace*)
VAR
	Sentence : STRING[30];
	NewSentence : STRING[20];
	FindWord : STRING[10];
	ReplaceWord : STRING[10];
	CmdFind : BOOL;
	SentenceLength : UDINT;
	NewSentenceLength : UDINT;
	NewSentenceSize : UDINT;
END_VAR
```

#### Main.st
```iecst
(*******************************************************************************
 * File       Sample\Main.st
 * Author:    Tyler Matijevich
 * Created:   September 27, 2020/11:19
********************************************************************************
 * Description: Example program for formatting string in IEC code and logging
 user entries in the logger
********************************************************************************)

PROGRAM _INIT

	// Initialize REAL and DINT variables
	VarDint 	:= 45678; // Try -2147483648
	VarReal 	:= 3.141592653589; // 32 bit floating value with more than enough significant digits, try -12345600000.0

	Size := SIZEOF(Message);

	// Runtime values
	FormatArgs.b[0] := FALSE; // BOOL
	FormatArgs.r[0] := 78.768; // LREAL
	FormatArgs.i[0] := -2144327918; // DINT, e.g. Status ID
	FormatArgs.s[0] := 'INIT'; // STRING

	Format := 'Status %b, Temp %r F, Code %i, State %s';

	MyNumber := -1234;
	Padding := 6;
	Spaces := TRUE;

END_PROGRAM

PROGRAM _CYCLIC

	// Test DINT and REAL to STRING conversions
	ReturnDint := brsitoa(VarDint, ADR(sDint));
	ReturnReal := brsftoa(VarReal, ADR(sReal));

	// The watch window will only print out 85 characters
	Length := IecFormatString(Message, Size, Format, FormatArgs);

	// Pad a number
	IecPadNumber(MyNumber, Number, Padding, Spaces);

END_PROGRAM

PROGRAM _EXIT

END_PROGRAM
```

### Program Logical/TestCStr

#### Main.c
```c
#include <bur/plc.h>
#include <string.h>
#include <stdint.h>

_LOCAL uint8_t a[11];
_LOCAL uint8_t b[21];

_LOCAL uint8_t num_copy _VAR_INIT(5);
_LOCAL uint8_t num_concat _VAR_INIT(5);

_LOCAL uint8_t copy;
_LOCAL uint8_t concat;
_LOCAL uint8_t init;

void _INIT ProgramInit(void)
{
	uint8_t i;

	for (i = 0; i < sizeof(a) - 1; i++)
		a[i] = i;
	a[sizeof(a) - 1] = 0;
}

void _CYCLIC ProgramCyclic(void)
{
	uint8_t i;

	if (copy) {
		copy = 0;
		strncpy((char*)a, (char*)b, num_copy);
	}

	if (concat) {
		concat = 0;
		strncat((char*)a, (char*)b, num_concat);
	}

	if (init) {
		init = 0;
		for (i = 0; i < sizeof(a) - 1; i++)
			a[i] = i;
		a[sizeof(a) - 1] = 0;
	}
}

void _EXIT ProgramExit(void)
{

}
```

### Program Logical/TestSuite (ANSIC)

#### main.c - Init, cyclic, exit code
```c
#ifdef _DEFAULT_INCLUDES
    #include <AsDefault.h>
#endif

#include <UnitTest.h>
#include <string.h>

UtMgrTestSuite_typ test_suite;

void _INIT ProgramInit(void)
{
    memset(&test_suite, 0, sizeof(test_suite));
    IecStringCopy(test_suite.Name, sizeof(test_suite.Name), "IecString_Tests");
    IecStringCopy(test_suite.Description, sizeof(test_suite.Description),
                "Test command and edges cases of all functions");
    test_suite.Type = utMgrTEST_TYPE_C;
    IecStringCopy(test_suite.MetaInformation,
                sizeof(test_suite.MetaInformation),
                "Test cases for IecString library");
    utInit(&test_suite);
}

void _CYCLIC ProgramCyclic(void)
{
    utCyclic(&test_suite);
}

void _EXIT ProgramExit(void)
{
    utExit(&test_suite);
}
```

#### load.c - Set loader and handler
```c
#include <UnitTest.h>

UNITTEST_TESTSET_DECLARATION copy_set;
UNITTEST_TESTSET_DECLARATION concat_set;

UNITTEST_TESTSET_FIXTURES (utTestSets)
{
    new_TestSet(copy_set),
    new_TestSet(concat_set)
};

UNTITTEST_TESTSET_HANDLER();
```

#### test_copy.c - Test IecStringCopy
```c
#ifdef _DEFAULT_INCLUDES
    #include <AsDefault.h>
#endif

#include <UnitTest.h>
#include <IecString.h>
#include <string.h>
#include <stdint.h>

_TEST copy_basic(void) {
    char a[81], b[81];
    int32_t status;

    strcpy(b, "Hello World!");

    status = IecStringCopy(a, sizeof(a), b);

    TEST_ASSERT_EQUAL_STRING("Hello World!", a);
    TEST_ASSERT_EQUAL_INT(0, status);

    TEST_DONE;
}

_TEST copy_null(void) {
    char a[81];
    int32_t status;

    strcpy(a, "Test");

    status = IecStringCopy(a, sizeof(a), NULL);

    TEST_ASSERT_EQUAL_STRING("Test", a);
    TEST_ASSERT_EQUAL_INT(IECSTRING_ERROR_NULL, status);

    TEST_DONE;
}

_TEST copy_size(void) {
    char a[81], b[81];
    int32_t status;

    strcpy(a, "Test");

    status = IecStringCopy(a, 0, b);

    TEST_ASSERT_EQUAL_STRING("Test", a);
    TEST_ASSERT_EQUAL_INT(IECSTRING_ERROR_SIZE, status);

    TEST_DONE;
}

_TEST copy_overlap(void) {
    char a[81];
    int32_t status;

    strcpy(a, "Test overlap");

    status = IecStringCopy(a, sizeof(a), a + 5);

    TEST_ASSERT_EQUAL_STRING("Test overlap", a);
    TEST_ASSERT_EQUAL_INT(IECSTRING_ERROR_OVERLAP, status);

    TEST_DONE;
}

_TEST copy_truncate(void) {
    char a[11], b[81];
    int32_t status;

    strcpy(b, "0123456789abc");

    status = IecStringCopy(a, sizeof(a), b);

    TEST_ASSERT_EQUAL_STRING("0123456789", a);
    TEST_ASSERT_EQUAL_INT(IECSTRING_WARNING_TRUNCATE, status);

    TEST_DONE;
}

UNITTEST_FIXTURES(fixtures) {
    new_TestFixture("IecStringCopy basic", copy_basic),
    new_TestFixture("IecStringCopy null", copy_null),
    new_TestFixture("IecStringCopy size", copy_size),
    new_TestFixture("IecStringCopy overlap", copy_overlap),
    new_TestFixture("IecStringCopy truncate", copy_truncate)
};

UNITTEST_CALLER_TEST (copy_set, "IecStringCopy test set", fixtures);
```

#### test_concat.c - Test IecStringConcat
```c
#include <UnitTest.h>
#include <IecString.h>
#include <string.h>
#include <stdint.h>

_TEST concat_basic(void) {
    char a[81], b[81];
    int32_t status;

    strcpy(a, "Hello");
    strcpy(b, " World!");

    status = IecStringConcat(a, sizeof(a), b);

    TEST_ASSERT_EQUAL_STRING("Hello World!", a);
    TEST_ASSERT_EQUAL_INT(0, status);

    TEST_DONE;
}

_TEST concat_null_source(void) {
    char a[81];
    int32_t status;

    strcpy(a, "Test");

    status = IecStringConcat(a, sizeof(a), NULL);

    TEST_ASSERT_EQUAL_STRING("Test", a);
    TEST_ASSERT_EQUAL_INT(IECSTRING_ERROR_NULL, status);

    TEST_DONE;
}

_TEST concat_null_destination(void) {
    char b[81];
    int32_t status;

    strcpy(b, "Test");

    status = IecStringConcat(NULL, 10, b);

    TEST_ASSERT_EQUAL_INT(IECSTRING_ERROR_NULL, status);

    TEST_DONE;
}

_TEST concat_size(void) {
    char a[81], b[81];
    int32_t status;

    strcpy(a, "Test");

    status = IecStringConcat(a, 0, b);

    TEST_ASSERT_EQUAL_STRING("Test", a);
    TEST_ASSERT_EQUAL_INT(IECSTRING_ERROR_SIZE, status);

    TEST_DONE;
}

_TEST concat_overlap(void) {
    char a[81];
    int32_t status;

    strcpy(a, "Test overlap");

    status = IecStringConcat(a, sizeof(a), a + 5);

    TEST_ASSERT_EQUAL_STRING("Test overlap", a);
    TEST_ASSERT_EQUAL_INT(IECSTRING_ERROR_OVERLAP, status);

    TEST_DONE;
}

_TEST concat_truncate(void) {
    char a[11], b[81];
    int32_t status;

    strcpy(a, "0123456");
    strcpy(b, "789abc");

    status = IecStringConcat(a, sizeof(a), b);

    TEST_ASSERT_EQUAL_STRING("0123456789", a);
    TEST_ASSERT_EQUAL_INT(IECSTRING_WARNING_TRUNCATE, status);

    TEST_DONE;
}

UNITTEST_FIXTURES(fixtures) {
    new_TestFixture("IecStringConcat basic", concat_basic),
    new_TestFixture("IecStringConcat null source", concat_null_source),
    new_TestFixture("IecStringConcat null destination", concat_null_destination),
    new_TestFixture("IecStringConcat size", concat_size),
    new_TestFixture("IecStringConcat overlap", concat_overlap),
    new_TestFixture("IecStringConcat truncate", concat_truncate)
};

UNITTEST_CALLER_TEST (concat_set, "IecStringConcat test set", fixtures);
```

#### test_replace.c - Test IecStringReplace
```c
#ifdef _DEFAULT_INCLUDES
    #include <AsDefault.h>
#endif

#include <UnitTest.h>
#include <IecString.h>
#include <string.h>
#include <stdint.h>

_TEST replace_basic(void) {
    char a[81], b[81], f[81], r[81];
    int32_t status;

    strcpy(b, "The quick brown fox");
    strcpy(f, "quick");
    strcpy(r, "slow");

    status = IecStringReplace(a, sizeof(a), f, r, b);

    TEST_ASSERT_EQUAL_STRING("The slow brown fox", a);
    TEST_ASSERT_EQUAL_INT(0, status);

    TEST_DONE;
}

_TEST replace_multiple(void) {
    char a[81], b[81], f[81], r[81];
    int32_t status;

    strcpy(b, "The quick brown fox");
    strcpy(f, " ");
    strcpy(r, "_");

    status = IecStringReplace(a, sizeof(a), f, r, b);

    TEST_ASSERT_EQUAL_STRING("The_quick_brown_fox", a);
    TEST_ASSERT_EQUAL_INT(0, status);

    TEST_DONE;
}

_TEST replace_null_source(void) {
    char a[81], f[81], r[81];
    int32_t status;

    strcpy(a, "Test");

    status = IecStringReplace(a, sizeof(a), f, r, NULL);

    TEST_ASSERT_EQUAL_STRING("Test", a);
    TEST_ASSERT_EQUAL_INT(IECSTRING_ERROR_NULL, status);

    TEST_DONE;
}

_TEST replace_null_find(void) {
    char a[81], b[81], r[81];
    int32_t status;

    strcpy(a, "Test");

    status = IecStringReplace(a, sizeof(a), NULL, r, b);

    TEST_ASSERT_EQUAL_STRING("Test", a);
    TEST_ASSERT_EQUAL_INT(IECSTRING_ERROR_NULL, status);

    TEST_DONE;
}

_TEST replace_null_replace(void) {
    char a[81], b[81], f[81];
    int32_t status;

    strcpy(a, "Test");

    status = IecStringReplace(a, sizeof(a), f, NULL, b);

    TEST_ASSERT_EQUAL_STRING("Test", a);
    TEST_ASSERT_EQUAL_INT(IECSTRING_ERROR_NULL, status);

    TEST_DONE;
}

_TEST replace_null_destination(void) {
    char b[81], f[81], r[81];
    int32_t status;

    status = IecStringReplace(NULL, 11, f, r, b);

    TEST_ASSERT_EQUAL_INT(IECSTRING_ERROR_NULL, status);

    TEST_DONE;
}

_TEST replace_size(void) {
    char a[81], b[81], f[81], r[81];
    int32_t status;

    strcpy(a, "Test");
    strcpy(b, "The quick brown fox");
    strcpy(f, "quick");
    strcpy(r, "slow");

    status = IecStringReplace(a, 0, f, r, b);

    TEST_ASSERT_EQUAL_STRING("Test", a);
    TEST_ASSERT_EQUAL_INT(IECSTRING_ERROR_SIZE, status);

    TEST_DONE;
}

_TEST replace_length(void) {
    char a[81], b[81], f[81], r[81];
    int32_t status;

    strcpy(a, "Test");
    strcpy(b, "The quick brown fox");
    strcpy(f, "The quick brown fox jumps");
    strcpy(r, "slow");

    status = IecStringReplace(a, sizeof(a), f, r, b);

    TEST_ASSERT_EQUAL_STRING("Test", a);
    TEST_ASSERT_EQUAL_INT(IECSTRING_ERROR_LENGTH, status);

    TEST_DONE;
}

_TEST replace_overlap_source(void) {
    char a[81], f[81], r[81];
    int32_t status;

    strcpy(a, "Test");

    status = IecStringReplace(a, sizeof(a), f, r, a + 1);

    TEST_ASSERT_EQUAL_STRING("Test", a);
    TEST_ASSERT_EQUAL_INT(IECSTRING_ERROR_OVERLAP, status);

    TEST_DONE;
}

_TEST replace_overlap_find(void) {
    char a[81], b[81], r[81];
    int32_t status;

    strcpy(a, "Test");

    status = IecStringReplace(a, sizeof(a), a + 1, r, b);

    TEST_ASSERT_EQUAL_STRING("Test", a);
    TEST_ASSERT_EQUAL_INT(IECSTRING_ERROR_OVERLAP, status);

    TEST_DONE;
}

_TEST replace_overlap_replace(void) {
    char a[81], b[81], f[81];
    int32_t status;

    strcpy(a, "Test");

    status = IecStringReplace(a, sizeof(a), f, a + 1, b);

    TEST_ASSERT_EQUAL_STRING("Test", a);
    TEST_ASSERT_EQUAL_INT(IECSTRING_ERROR_OVERLAP, status);

    TEST_DONE;
}

_TEST replace_truncate(void) {
    char a[11], b[81], f[81], r[81];
    int32_t status;

    strcpy(b, "The quick brown fox");
    strcpy(f, "quick");
    strcpy(r, "slow");

    status = IecStringReplace(a, sizeof(a), f, r, b);

    TEST_ASSERT_EQUAL_STRING("The slow b", a);
    TEST_ASSERT_EQUAL_INT(IECSTRING_WARNING_TRUNCATE, status);

    TEST_DONE;
}

UNITTEST_FIXTURES(fixtures) {
    new_TestFixture("IecStringReplace basic", replace_basic),
    new_TestFixture("IecStringReplace multiple", replace_multiple),
    new_TestFixture("IecStringReplace null source", replace_null_source),
    new_TestFixture("IecStringReplace null find", replace_null_find),
    new_TestFixture("IecStringReplace null replace", replace_null_replace),
    new_TestFixture("IecStringReplace null destination", replace_null_destination),
    new_TestFixture("IecStringReplace size", replace_size),
    new_TestFixture("IecStringReplace length", replace_length),
    new_TestFixture("IecStringReplace overlap source", replace_overlap_source),
    new_TestFixture("IecStringReplace overlap find", replace_overlap_find),
    new_TestFixture("IecStringReplace overlap replace", replace_overlap_replace),
    new_TestFixture("IecStringReplace truncate", replace_truncate)
};

UNITTEST_CALLER_TEST (replace_set, "IecStringReplace test set", fixtures);
```

#### test_format.c - Test IecStringFormat
```c
#include <UnitTest.h>
#include <IecString.h>
#include <string.h>
#include <stdint.h>
#include <stdbool.h>

_TEST format_basic(void) {
    char a[81], b[81];
    IecStringFormatType args;
    int32_t status;

    strcpy(b, "Error: %b, Temp: %f C, Step: %i, Message: %s");
    args.b[0] = true;
    args.f[0] = 123.456;
    args.i[0] = 15;
    strcpy(args.s[0], "All clear");

    status = IecStringFormat(a, sizeof(a), b, &args);

    TEST_ASSERT_EQUAL_STRING("Error: TRUE, Temp: 123.456 C, Step: 15, Message: All clear", a);
    TEST_ASSERT_EQUAL_INT(0, status);

    TEST_DONE;
}

_TEST format_bool(void) {
    char a[81], b[81];
    IecStringFormatType args;
    int32_t status;

    strcpy(b, "%b %b %b %b %b %b %b");
    memset(args.b, 0, sizeof(args.b));
    args.b[1] = true;

    status = IecStringFormat(a, sizeof(a), b, &args);

    TEST_ASSERT_EQUAL_STRING("FALSE TRUE FALSE FALSE FALSE FALSE ", a);
    TEST_ASSERT_EQUAL_INT(0, status);

    TEST_DONE;
}

_TEST format_double(void) {
    char a[81], b[81];
    IecStringFormatType args;
    int32_t status;

    strcpy(b, "%f, %f, %f, %f");
    args.f[0] = -123;
    args.f[1] = 0.0456;
    args.f[2] = 12e7;
    args.f[3] = 123456789;

    status = IecStringFormat(a, sizeof(a), b, &args);

    TEST_ASSERT_EQUAL_STRING("-123, 0.0456, 1.2e+08, 1.23457e+08", a);
    TEST_ASSERT_EQUAL_INT(0, status);

    TEST_DONE;
}

_TEST format_int(void) {
    char a[81], b[81];
    IecStringFormatType args;
    int32_t status;

    strcpy(b, "%i, %i, %i, %i, %i");
    args.i[0] = -123;
    args.i[1] = INT32_MAX;
    args.i[2] = INT32_MIN;
    args.i[3] = UINT32_MAX;
    args.i[4] = 2147483648U;

    status = IecStringFormat(a, sizeof(a), b, &args);

    TEST_ASSERT_EQUAL_STRING("-123, 2147483647, -2147483648, -1, -2147483648", a);
    TEST_ASSERT_EQUAL_INT(0, status);

    TEST_DONE;
}

_TEST format_string(void) {
    char a[81], b[81];
    IecStringFormatType args;
    int32_t status;

    strcpy(b, "%s, %s, %s");
    strcpy(args.s[0], "one");
    strcpy(args.s[1], "two");
    strcpy(args.s[2], "three");

    status = IecStringFormat(a, sizeof(a), b, &args);

    TEST_ASSERT_EQUAL_STRING("one, two, three", a);
    TEST_ASSERT_EQUAL_INT(0, status);

    TEST_DONE;
}

_TEST format_null_source(void) {
    char a[81];
    IecStringFormatType args;
    int32_t status;

    strcpy(a, "Test");

    status = IecStringFormat(a, sizeof(a), NULL, &args);

    TEST_ASSERT_EQUAL_STRING("Test", a);
    TEST_ASSERT_EQUAL_INT(IECSTRING_ERROR_NULL, status);

    TEST_DONE;
}

_TEST format_null_destination(void) {
    char b[81];
    IecStringFormatType args;
    int32_t status;

    strcpy(b, "Test");

    status = IecStringFormat(NULL, 10, b, &args);

    TEST_ASSERT_EQUAL_INT(IECSTRING_ERROR_NULL, status);

    TEST_DONE;
}

_TEST format_null_values(void) {
    char a[81], b[81];
    int32_t status;

    strcpy(a, "Test");

    status = IecStringFormat(a, sizeof(a), b, NULL);

    TEST_ASSERT_EQUAL_STRING("Test", a);
    TEST_ASSERT_EQUAL_INT(IECSTRING_ERROR_NULL, status);

    TEST_DONE;
}

_TEST format_size(void) {
    char a[81], b[81];
    IecStringFormatType args;
    int32_t status;

    strcpy(a, "Test");

    status = IecStringFormat(a, 0, b, &args);

    TEST_ASSERT_EQUAL_STRING("Test", a);
    TEST_ASSERT_EQUAL_INT(IECSTRING_ERROR_SIZE, status);

    TEST_DONE;
}

_TEST format_overlap(void) {
    char a[81];
    IecStringFormatType args;
    int32_t status;

    strcpy(a, "Test overlap");

    status = IecStringFormat(a, sizeof(a), a + 5, &args);

    TEST_ASSERT_EQUAL_STRING("Test overlap", a);
    TEST_ASSERT_EQUAL_INT(IECSTRING_ERROR_OVERLAP, status);

    TEST_DONE;
}

_TEST format_truncate(void) {
    char a[11], b[81];
    IecStringFormatType args;
    int32_t status;

    strcpy(b, "%s, %s, %s");
    strcpy(args.s[0], "one");
    strcpy(args.s[1], "two");
    strcpy(args.s[2], "three");

    status = IecStringFormat(a, sizeof(a), b, &args);

    TEST_ASSERT_EQUAL_STRING("one, two, ", a);
    TEST_ASSERT_EQUAL_INT(IECSTRING_WARNING_TRUNCATE, status);

    TEST_DONE;
}

UNITTEST_FIXTURES(fixtures) {
    new_TestFixture("IecStringFormat basic", format_basic),
    new_TestFixture("IecStringFormat bool", format_bool),
    new_TestFixture("IecStringFormat double", format_double),
    new_TestFixture("IecStringFormat int", format_int),
    new_TestFixture("IecStringFormat string", format_string),
    new_TestFixture("IecStringFormat null source", format_null_source),
    new_TestFixture("IecStringFormat null destination", format_null_destination),
    new_TestFixture("IecStringFormat null values", format_null_values),
    new_TestFixture("IecStringFormat size", format_size),
    new_TestFixture("IecStringFormat overlap", format_overlap),
    new_TestFixture("IecStringFormat truncate", format_truncate)
};

UNITTEST_CALLER_TEST (format_set, "IecStringFormat test set", fixtures);
```

#### test_pad.c - Test IecStringPadInt
```c
#include <UnitTest.h>
#include <IecString.h>
#include <string.h>
#include <stdint.h>

_TEST padint_zeros(void) {
    char a[81];
    int32_t number, status;

    number = 1234;

    status = IecStringPadInt(a, sizeof(a), number, 6, 0);

    TEST_ASSERT_EQUAL_STRING("001234", a);
    TEST_ASSERT_EQUAL_INT(0, status);

    TEST_DONE;
}

_TEST padint_spaces(void) {
    char a[81];
    int32_t number, status;

    number = -5678;

    status = IecStringPadInt(a, sizeof(a), number, 6, 1);

    TEST_ASSERT_EQUAL_STRING("-  5678", a);
    TEST_ASSERT_EQUAL_INT(0, status);

    TEST_DONE;
}

_TEST padint_max(void) {
    char a[81];
    int32_t number, status;

    number = INT32_MAX;

    status = IecStringPadInt(a, sizeof(a), number, 0, 0);

    TEST_ASSERT_EQUAL_STRING("2147483647", a);
    TEST_ASSERT_EQUAL_INT(0, status);

    TEST_DONE;
}

_TEST padint_min(void) {
    char a[81];
    int32_t number, status;

    number = INT32_MIN;

    status = IecStringPadInt(a, sizeof(a), number, 0, 0);

    TEST_ASSERT_EQUAL_STRING("-2147483648", a);
    TEST_ASSERT_EQUAL_INT(0, status);

    TEST_DONE;
}

_TEST padint_size(void) {
    char a[6];
    int32_t number, status;

    strcpy(a, "abc");
    number = 123456;

    status = IecStringPadInt(a, sizeof(a), number, 0, 0);

    TEST_ASSERT_EQUAL_STRING("abc", a);
    TEST_ASSERT_EQUAL_INT(IECSTRING_ERROR_SIZE, status);

    TEST_DONE;
}

_TEST padint_null(void) {
    int32_t number, status;

    number = 123456;

    status = IecStringPadInt(NULL, 7, number, 0, 0);

    TEST_ASSERT_EQUAL_INT(IECSTRING_ERROR_NULL, status);

    TEST_DONE;
}

UNITTEST_FIXTURES(fixtures) {
    new_TestFixture("IecStringPadInt zeros", padint_zeros),
    new_TestFixture("IecStringPadInt spaces", padint_spaces),
    new_TestFixture("IecStringPadInt max", padint_max),
    new_TestFixture("IecStringPadInt min", padint_min),
    new_TestFixture("IecStringPadInt size error", padint_size),
    new_TestFixture("IecStringPadInt null error", padint_null)
};

UNITTEST_CALLER_TEST (padint_set, "IecStringPadInt test set", fixtures);
```

#### Variables.var - not listed in the package file held
```iecst
VAR
	TestSuite : UtMgrTestSuite;
END_VAR
```

#### Loader.c - not listed in the package file held
```c
#include <UnitTest.h>

UNITTEST_TESTSET_DECLARATION copy_set;

UNITTEST_TESTSET_FIXTURES (utTestSets)
{
	new_TestSet(copy_set)
};

UNTITTEST_TESTSET_HANDLER();
```

#### test_integer.c - not listed in the package file held
```c
#include <UnitTest.h>
#include <IecString.h>
#include <string.h>
#include <stdint.h>

_TEST integer_zeros(void) {
    char a[81];
    int32_t number, status;

    number = 1234;

    status = IecStringInteger(a, sizeof(a), number, 6, 0);

    TEST_ASSERT_EQUAL_STRING("001234", a);
    TEST_ASSERT_EQUAL_INT(0, status);

    TEST_DONE;
}

_TEST integer_spaces(void) {
    char a[81];
    int32_t number, status;

    number = -5678;

    status = IecStringInteger(a, sizeof(a), number, 6, 1);

    TEST_ASSERT_EQUAL_STRING("-  5678", a);
    TEST_ASSERT_EQUAL_INT(0, status);

    TEST_DONE;
}

_TEST integer_max(void) {
    char a[81];
    int32_t number, status;

    number = INT32_MAX;

    status = IecStringInteger(a, sizeof(a), number, 0, 0);

    TEST_ASSERT_EQUAL_STRING("2147483647", a);
    TEST_ASSERT_EQUAL_INT(0, status);

    TEST_DONE;
}

_TEST integer_min(void) {
    char a[81];
    int32_t number, status;

    number = INT32_MIN;

    status = IecStringInteger(a, sizeof(a), number, 0, 0);

    TEST_ASSERT_EQUAL_STRING("-2147483648", a);
    TEST_ASSERT_EQUAL_INT(0, status);

    TEST_DONE;
}

_TEST integer_size(void) {
    char a[6];
    int32_t number, status;

    strcpy(a, "abc");
    number = 123456;

    status = IecStringInteger(a, sizeof(a), number, 0, 0);

    TEST_ASSERT_EQUAL_STRING("abc", a);
    TEST_ASSERT_EQUAL_INT(IECSTRING_ERROR_SIZE, status);

    TEST_DONE;
}

_TEST integer_null(void) {
    int32_t number, status;

    number = 123456;

    status = IecStringInteger(NULL, 7, number, 0, 0);

    TEST_ASSERT_EQUAL_INT(IECSTRING_ERROR_NULL, status);

    TEST_DONE;
}

UNITTEST_FIXTURES(fixtures) {
    new_TestFixture("IecStringInteger zeros", integer_zeros),
    new_TestFixture("IecStringInteger spaces", integer_spaces),
    new_TestFixture("IecStringInteger max", integer_max),
    new_TestFixture("IecStringInteger min", integer_min),
    new_TestFixture("IecStringInteger size error", integer_size),
    new_TestFixture("IecStringInteger null error", integer_null)
};

UNITTEST_CALLER_TEST (integer_set, "IecStringInteger test set", fixtures);
```

#### TestCopy.c - not listed in the package file held
```c
#include <bur/plctypes.h>

#ifdef _DEFAULT_INCLUDES
	#include <AsDefault.h>
#endif

#include <UnitTest.h>
#include <IecString.h>
#include <string.h>
#include <stdint.h>

_TEST copy_basic (void)
{
	char string1[81], string2[81];
	uint32_t return_value;

	memset(string1, 0, sizeof(string1));
	strcpy(string2, "Hello World!");

	return_value = IecStringCopy(string1, string2, sizeof(string1));

	TEST_ASSERT_EQUAL_STRING("Hello World!", string1);
	TEST_ASSERT_EQUAL_INT((uint32_t)&string1, return_value);

	TEST_DONE;
}

_TEST copy_null (void)
{
	char string1[81], string2[81];
	uint32_t return_value;

	memset(string1, 0, sizeof(string1));

	return_value = IecStringCopy(string1, NULL, sizeof(string1));

	/* Return destination and do not write to destination */
	TEST_ASSERT_EQUAL_STRING("", string1);
	TEST_ASSERT_EQUAL_INT((uint32_t)&string1, return_value);

	return_value = IecStringCopy(NULL, string2, sizeof(string1));

	/* Return destination even if null */
	TEST_ASSERT_EQUAL_INT(NULL, return_value);

	TEST_DONE;
}

_TEST copy_zero (void)
{
	char string1[81], string2[81];
	uint32_t return_value;

	strcpy(string1, "Test");
	strcpy(string2, "Zero");

	return_value = IecStringCopy(string1, string2, 0);

	/* Abort copy if size is zero and do not write to destination */
	TEST_ASSERT_EQUAL_STRING("Test", string1);
	TEST_ASSERT_EQUAL_INT((uint32_t)&string1, return_value);

	TEST_DONE;
}

_TEST copy_one (void)
{
	char string1[81], string2[81];

	strcpy(string1, "Test");
	strcpy(string2, "Zero");

	IecStringCopy(string1, string2, 1);

	/* Copy one null character */
	TEST_ASSERT_EQUAL_STRING("", string1);

	TEST_DONE;
}

_TEST copy_partial (void)
{
	char string1[81], string2[81];

	memset(string1, 0, sizeof(string1));
	strcpy(string2, "Hello World!");

	IecStringCopy(string1, string2, 6);

	TEST_ASSERT_EQUAL_STRING("Hello", string1);

	TEST_DONE;
}

_TEST copy_overflow (void)
{
	char string1[6], string2[11];

	memset(string1, 0, sizeof(string1));
	strcpy(string2, "IecString");

	IecStringCopy(string1, string2, sizeof(string1));

	TEST_ASSERT_EQUAL_STRING("IecSt", string1);

	TEST_DONE;
}

UNITTEST_FIXTURES (fixtures)
{
	new_TestFixture("IecStringCopy basic", copy_basic),
	new_TestFixture("IecStringCopy null", copy_null),
	new_TestFixture("IecStringCopy zero", copy_zero),
	new_TestFixture("IecStringCopy one", copy_one),
	new_TestFixture("IecStringCopy partial", copy_partial),
	new_TestFixture("IecStringCopy overflow", copy_overflow)
};

UNITTEST_CALLER_TEST (copy_set, "IecStringCopy test set", fixtures);
```

Listed in the project but not available here: Logical/Source/UnitTest/TestSuite/main.c, Logical/Source/Compare/TestCStr
